(* CoDeSys 2.3.9.37 project: Cap5_5_Res.pro *)
(* Libraries: Standard.lib 4.10.05 12:14:46 *)

(* Global variable list: Global_Variables *)
VAR_GLOBAL
  (* Entradas *)
  Boton : BOOL;
  BotonReset: BOOL;
  (* Salida *)
  Valor : INT;
END_VAR

(* POU PLC_PRG, ST *)
PROGRAM PLC_PRG
VAR
    MiContador : Contador;
END_VAR
MiContador(Entrada:=Boton, Reset:=BotonReset, Salida=>Valor);
END_PROGRAM

(* POU Contador, ST *)
FUNCTION_BLOCK Contador
VAR_INPUT
   Entrada: BOOL;
   Reset: BOOL;
END_VAR
VAR_OUTPUT
   Salida : INT;
END_VAR
VAR
   Detector :DeteccionFlanco ;
    Pulso: BOOL;
END_VAR
Detector(CLK:=Entrada, Q=>Pulso);
IF Reset=TRUE THEN
   Salida:=0;
ELSE
  IF Pulso=TRUE THEN
        Salida:=Salida+1;
  END_IF
END_IF
END_FUNCTION_BLOCK

(* POU DeteccionFlanco, LD *)
FUNCTION_BLOCK DeteccionFlanco
VAR_INPUT
    CLK: BOOL;
END_VAR
VAR_OUTPUT
    Q: BOOL;
END_VAR
VAR
   CLK_OLD:BOOL:=FALSE;
END_VAR
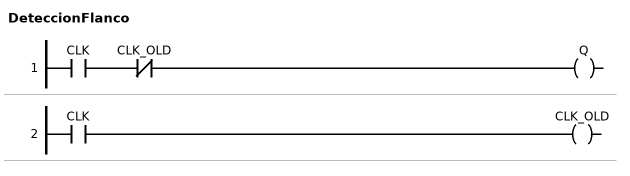
_LD_ (* Ladder Diagram *)
NETWORK 1
	[CLK] - [/CLK_OLD] --- (Q)
NETWORK 2
	[CLK] --- (CLK_OLD)
_END_LD_
(* the same logic as Structured Text *)
(* Network 1 *)
Q := CLK AND NOT CLK_OLD;
(* Network 2 *)
CLK_OLD := CLK;
END_FUNCTION_BLOCK

(* Visualisation Visu
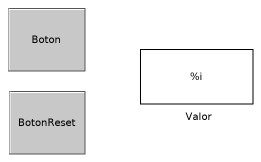
button at (30,50)-(107,113): text "Boton"; taps Boton
button at (31,133)-(107,196): text "BotonReset"; taps BotonReset
rectangle at (162,91)-(275,146): text "%i"; shows Valor
rectangle at (177,146)-(264,171): text "Valor"
*)
